FUNCTION LongStringLen : UDINT
VAR_INPUT
	In : ANY_STRING;
END_VAR
VAR
	i : UDINT;
END_VAR

IF NOT In.TypeClass = __SYSTEM.TYPE_CLASS.TYPE_STRING THEN
	RETURN;
END_IF

WHILE (In.pValue[i] <> 0) DO
	i := i+1;
END_WHILE

LongStringLen := i;

END_FUNCTION

(* stored: Version 1.1.0.1, ProductVersion 3.1.4024.12
   POU LongStringLen: Id {75af9dd5-a27d-04b1-199a-a3624449c9b9}, SpecialFunc None *)
